Universal Robots PolyScope program: MixerToLocal.urp

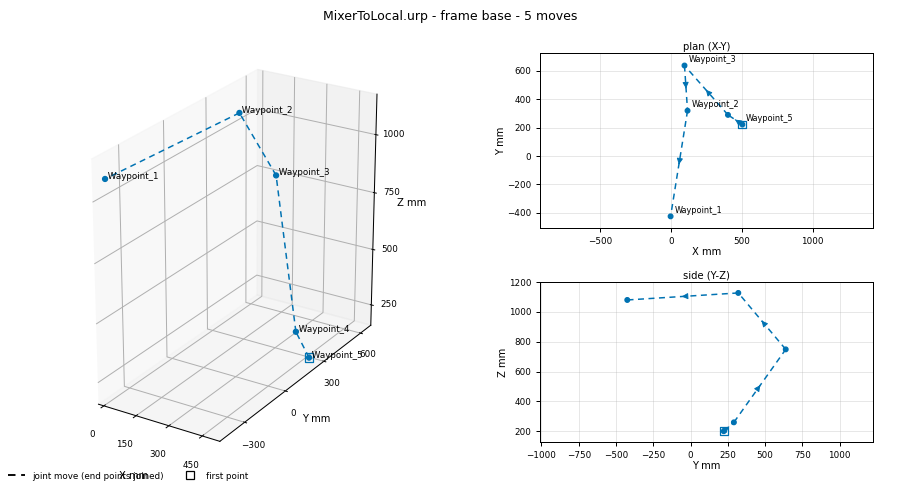
[picture p0: tool path of MixerToLocal.urp in frame base, 5 of 5 moves have a stored position in this frame; points joined in program order, loops and branches not executed]
Program MixerToLocal (installation=Youssef directory=/programs/Youssef createdIn=5.9.5.1031259 lastSavedIn=5.9.5.1031259 robotSerialNumber=20215500597)
Calibrated DH parameters: a=[0.000193, -0.066673, -0.391568, -0.000012, 0.00005, 0]; d=[0.162643, -472.05677, 465.132521, 7.058239, 0.099746, 0.099582]; alpha=[1.571116, 0.00089, 0.003862, 1.569269, -1.569248, 0]; deltaTheta=[0, -1.413394, 7.628392, 0.068187, 0, -0.000001]
Robot Program (runOnlyOnce=true)
  MoveJ speed 60 deg/s, acceleration 80 deg/s^2 (useActiveTCP=true) feature=Base
    Waypoint Waypoint_5: TCP in base x=504.233 y=222.177 z=200.516 mm, rx=1.2172 ry=1.1583 rz=1.214 rad; joints [72.581, -92.271, -136.674, -125.916, -15.588, -3.757] deg; TCP offset x=0 y=0 z=191.5 mm, rx=0 ry=0 rz=0 rad
    Waypoint Waypoint_4: TCP in base x=402.516 y=290.095 z=259.958 mm, rx=1.3002 ry=1.1489 rz=1.2399 rad; joints [94.435, -83.523, -131.099, -136.444, 6.698, -3.896] deg
    Waypoint Waypoint_3: TCP in base x=96.27 y=637.775 z=749.236 mm, rx=-1.4855 ry=-0.0307 rz=0.0319 rad; joints [94.292, -84.133, -90.199, -0.883, 88.027, -0.054] deg
    Waypoint Waypoint_2: TCP in base x=117.665 y=319.704 z=1127.649 mm, rx=-1.3628 ry=-0.0281 rz=0.0448 rad; joints [94.93, -84.768, -17.496, -65.907, 88.027, -0.059] deg
    Waypoint Waypoint_1: TCP in base x=-1.655 y=-424.817 z=1080.554 mm, rx=-0.0046 ry=-2.2185 rz=2.2204 rad; joints [-0.002, -89.996, 0.002, -89.996, -0.002, -0.002] deg
